(* IEC 61131-3 sources: SmartHomeNew/workspace/dut_rebuild/alarm, 5 files *)

(* ---- ST_Alarm_Core_Record_V2.dut ---- *)
TYPE ST_Alarm_Core_Record_V2 :
STRUCT
    id : UDINT;
    timestamp_ms : UDINT;
    source_code : UINT;
    source_instance : UINT;
    severity : E_ALERT_PRIORITY;
    is_active : BOOL;
    is_acknowledged : BOOL;
    cause_code : UINT;
END_STRUCT
END_TYPE

(* ---- ST_Alarm_View_Record_V2.dut ---- *)
TYPE ST_Alarm_View_Record_V2 :
STRUCT
    core : ST_Alarm_Core_Record_V2;
    source_text : STRING(32);
    message_text : STRING(200);
END_STRUCT
END_TYPE

(* ---- FB_Alarm_Compatibility_Package_DRAFT.st ---- *)
FUNCTION_BLOCK FB_Alarm_Compatibility_Package_DRAFT
VAR_INPUT
    VI_Alarm_Legacy : ST_Alarm;
END_VAR
VAR_OUTPUT
    VO_Alarm_Legacy_Roundtrip : ST_Alarm;
    VO_OK : BOOL;
END_VAR
VAR
    fbFwd : FB_Alarm_Legacy_To_V2_Adapter_DRAFT;
    fbRev : FB_Alarm_V2_To_Legacy_Adapter_DRAFT;
    L_Temp_V2 : ST_Alarm_V2;
END_VAR

fbFwd(VI_Alarm_Legacy := VI_Alarm_Legacy, VO_Alarm_V2 => L_Temp_V2, VO_Translation_OK => VO_OK);
fbRev(VI_Alarm_V2 := L_Temp_V2, VO_Alarm_Legacy => VO_Alarm_Legacy_Roundtrip);

END_FUNCTION_BLOCK

(* ---- FB_Alarm_Legacy_To_V2_Adapter_DRAFT.st ---- *)
FUNCTION_BLOCK FB_Alarm_Legacy_To_V2_Adapter_DRAFT
VAR_INPUT
    VI_Alarm_Legacy : ST_Alarm;
END_VAR
VAR_OUTPUT
    VO_Alarm_V2 : ST_Alarm_V2;
    VO_Translation_OK : BOOL;
END_VAR

VO_Alarm_V2.id := VI_Alarm_Legacy.id;
VO_Alarm_V2.enabled := VI_Alarm_Legacy.enabled;
VO_Alarm_V2.severity := VI_Alarm_Legacy.severity;
VO_Alarm_V2.source_id := VI_Alarm_Legacy.source_id;
VO_Alarm_V2.active := VI_Alarm_Legacy.active;

VO_Translation_OK := TRUE;
END_FUNCTION_BLOCK

(* ---- FB_Alarm_V2_To_Legacy_Adapter_DRAFT.st ---- *)
FUNCTION_BLOCK FB_Alarm_V2_To_Legacy_Adapter_DRAFT
VAR_INPUT
    VI_Alarm_V2 : ST_Alarm_V2;
END_VAR
VAR_OUTPUT
    VO_Alarm_Legacy : ST_Alarm;
    VO_Translation_OK : BOOL;
END_VAR

VO_Alarm_Legacy.id := VI_Alarm_V2.id;
VO_Alarm_Legacy.enabled := VI_Alarm_V2.enabled;
VO_Alarm_Legacy.severity := VI_Alarm_V2.severity;
VO_Alarm_Legacy.source_id := VI_Alarm_V2.source_id;
VO_Alarm_Legacy.active := VI_Alarm_V2.active;

VO_Translation_OK := TRUE;
END_FUNCTION_BLOCK
